// TIA Portal V18 export
FUNCTION_BLOCK "Stacklight"   // FB20, LAD
TITLE = Description:
{ S7_Optimized_Access := 'TRUE' }
VERSION : 0.1
// The stacklight is showing the status of the machine and checking different conditions:
// - errors from the drives (PLC)
// - communication (NOAH)
// - errors from the fluid supply (NOAH)
// - doors (PLC)
// 
// RED - default color, error or PLC is turning on
// ORANGE - door open or in maintenance mode
// GREEN - machine connected and working fine
// 
// RED-GREEN blinking - machine ready to connect
// 
// Date:
// stored: AutoNumber true, IsIECCheckEnabled false, IsRetainMemResEnabled false, MemoryReserve 100, SetENOAutomatically false, UDAEnableTagReadback false
   VAR_INPUT
      Emergency : Bool;
      Mode : Int;
      RedIn : Bool;
      YellowIn : Bool;
      GreenIn : Bool;
      ReadyDevices : Bool;
      DoorOpen : Bool;
      Xvelocity : DInt;
      Yvelocity : DInt;
      MachineReadyPLC : Bool;
      MachineReadyNOAH : Bool;
      MachinePrintingPLC : Bool;
      MachinePrintingNOAH : Bool;
      MachineErrorPLC : Bool;
      MachineErrorNOAH : Bool;
      LED01 : Bool;
      LED02 : Bool;
      Maintenance : Int;
   END_VAR
   VAR_OUTPUT
      Status : Int;
      OutputColor : Int;
      StacklightCTRL01 : Bool;
      StacklightCTRL02 : Bool;
   END_VAR
   VAR_IN_OUT
      MachineConnectedNOAH : Bool;
   END_VAR
   VAR
      TriggerVelocityForMoving : DInt := 5;
      GreenInternal : Bool;
      YellowInternal : Bool;
      RedInternal : Bool;
      ColorInternal : Int;   // 0 = Red; 1 = Orange; 2 = Green;
      MachineMovingInternal : Bool;
      MachineConnectedPLC : Bool;
      MachineConnectedInternal : Bool;
   END_VAR
   VAR CONSTANT
      MachineConnectedWaitTime : Time := T#3s;
      MachineConnectedResetTime : Time := T#200ms;
   END_VAR
BEGIN

REGION Network 1: Machine Moving Status Read
   // Checking if the machine is moving.
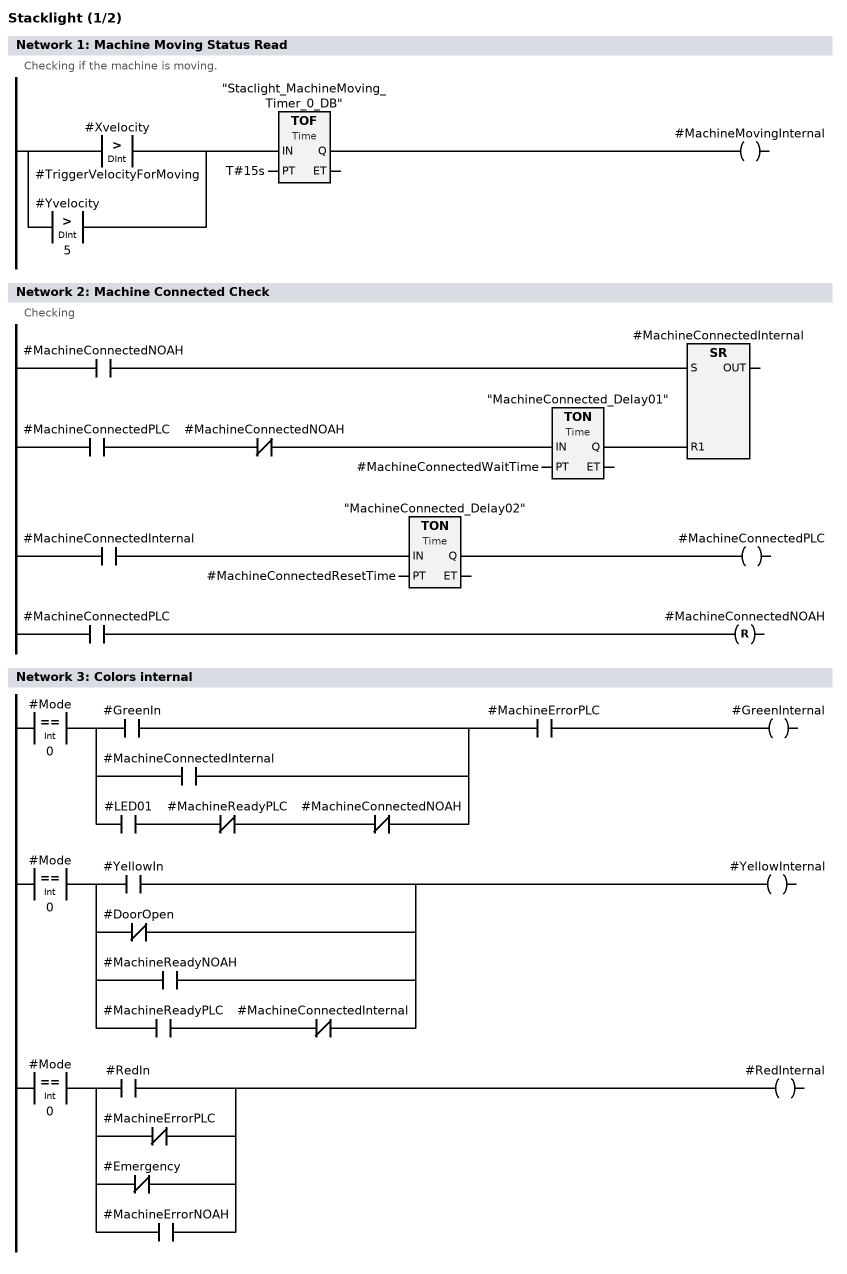
   RUNG wire#powerrail
      { S7_Templates := "SrcType := DInt" } GT_Contact(in1 := #Xvelocity, in2 := #TriggerVelocityForMoving)
      wire#w1
      { S7_Templates := "time_type := Time" } "Staclight_MachineMoving_Timer_0_DB".TOF(pt := T#15s, et =>)
      Coil( #MachineMovingInternal )
   END_RUNG
   RUNG wire#powerrail
      { S7_Templates := "SrcType := DInt" } GT_Contact(in1 := #Yvelocity, in2 := 5)
   END_RUNG wire#w1
   // the same network as SCL:
   "Staclight_MachineMoving_Timer_0_DB".TOF(IN := (#Xvelocity > #TriggerVelocityForMoving) OR (#Yvelocity > 5),
                           PT := T#15s);
   #MachineMovingInternal := "Staclight_MachineMoving_Timer_0_DB".Q;
END_REGION

REGION Network 2: Machine Connected Check
   // Checking
   RUNG wire#powerrail
      Contact( #MachineConnectedNOAH )
      S_SR(operand := #MachineConnectedInternal, r1 := wire#w1)
   END_RUNG
   RUNG wire#powerrail
      Contact( #MachineConnectedPLC )
      I_Contact( #MachineConnectedNOAH )
      { S7_Templates := "time_type := Time" } "MachineConnected_Delay01".TON(pt := #MachineConnectedWaitTime, et =>)
   END_RUNG wire#w1
   RUNG wire#powerrail
      Contact( #MachineConnectedInternal )
      { S7_Templates := "time_type := Time" } "MachineConnected_Delay02".TON(pt := #MachineConnectedResetTime, et =>)
      Coil( #MachineConnectedPLC )
   END_RUNG
   RUNG wire#powerrail
      Contact( #MachineConnectedPLC )
      R_Coil( #MachineConnectedNOAH )
   END_RUNG
   // the same network as SCL:
   "MachineConnected_Delay01".TON(IN := #MachineConnectedPLC AND NOT #MachineConnectedNOAH,
                           PT := #MachineConnectedWaitTime);
   IF #MachineConnectedNOAH THEN
       #MachineConnectedInternal := TRUE;   // SR flip-flop
   END_IF;
   IF "MachineConnected_Delay01".Q THEN #MachineConnectedInternal := FALSE; END_IF;
   "MachineConnected_Delay02".TON(IN := #MachineConnectedInternal, PT := #MachineConnectedResetTime);
   #MachineConnectedPLC := "MachineConnected_Delay02".Q;
   IF #MachineConnectedPLC THEN #MachineConnectedNOAH := FALSE; END_IF;
END_REGION

REGION Network 3: Colors internal
   RUNG wire#powerrail
      { S7_Templates := "SrcType := Int" } EQ_Contact(in1 := #Mode, in2 := 0)
      wire#w1
      Contact( #GreenIn )
      wire#w2
      Contact( #MachineErrorPLC )
      Coil( #GreenInternal )
   END_RUNG
   RUNG wire#w1
      Contact( #MachineConnectedInternal )
   END_RUNG wire#w2
   RUNG wire#w1
      Contact( #LED01 )
      I_Contact( #MachineReadyPLC )
      I_Contact( #MachineConnectedNOAH )
   END_RUNG wire#w2
   RUNG wire#powerrail
      { S7_Templates := "SrcType := Int" } EQ_Contact(in1 := #Mode, in2 := 0)
      wire#w3
      Contact( #YellowIn )
      wire#w4
      Coil( #YellowInternal )
   END_RUNG
   RUNG wire#w3
      I_Contact( #DoorOpen )
   END_RUNG wire#w4
   RUNG wire#w3
      Contact( #MachineReadyNOAH )
   END_RUNG wire#w4
   RUNG wire#w3
      Contact( #MachineReadyPLC )
      I_Contact( #MachineConnectedInternal )
   END_RUNG wire#w4
   RUNG wire#powerrail
      { S7_Templates := "SrcType := Int" } EQ_Contact(in1 := #Mode, in2 := 0)
      wire#w5
      Contact( #RedIn )
      wire#w6
      Coil( #RedInternal )
   END_RUNG
   RUNG wire#w5
      I_Contact( #MachineErrorPLC )
   END_RUNG wire#w6
   RUNG wire#w5
      I_Contact( #Emergency )
   END_RUNG wire#w6
   RUNG wire#w5
      Contact( #MachineErrorNOAH )
   END_RUNG wire#w6
   // the same network as SCL:
   #GreenInternal := (#Mode = 0) AND (#GreenIn OR #MachineConnectedInternal OR (#LED01 AND NOT #MachineReadyPLC AND NOT #MachineConnectedNOAH)) AND #MachineErrorPLC;
   #YellowInternal := (#Mode = 0) AND (#YellowIn OR NOT #DoorOpen OR #MachineReadyNOAH OR (#MachineReadyPLC AND NOT #MachineConnectedInternal));
   #RedInternal := (#Mode = 0) AND (#RedIn OR NOT #MachineErrorPLC OR NOT #Emergency OR #MachineErrorNOAH);
END_REGION

REGION Network 4: Status Move
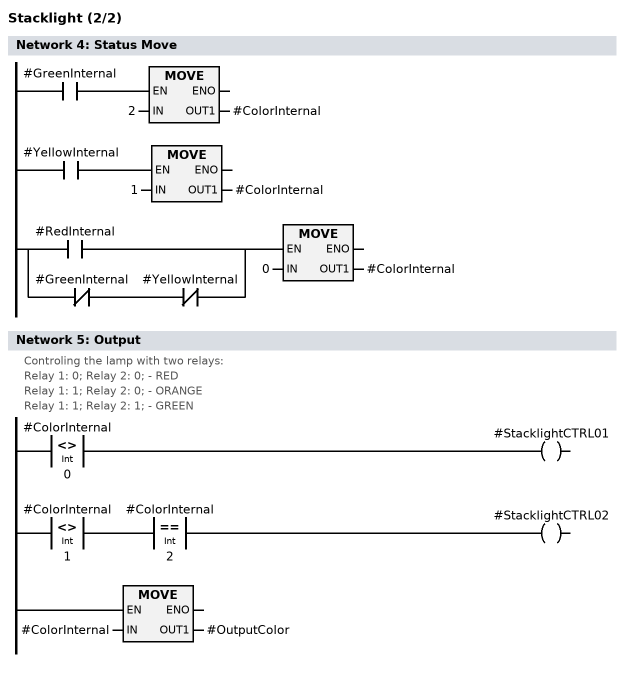
   RUNG wire#powerrail
      Contact( #GreenInternal )
      Move(in := 2, out1 => #ColorInternal)
   END_RUNG
   RUNG wire#powerrail
      Contact( #YellowInternal )
      Move(in := 1, out1 => #ColorInternal)
   END_RUNG
   RUNG wire#powerrail
      Contact( #RedInternal )
      wire#w1
      Move(in := 0, out1 => #ColorInternal)
   END_RUNG
   RUNG wire#powerrail
      I_Contact( #GreenInternal )
      I_Contact( #YellowInternal )
   END_RUNG wire#w1
   // the same network as SCL:
   IF #GreenInternal THEN #ColorInternal := 2; END_IF;
   IF #YellowInternal THEN #ColorInternal := 1; END_IF;
   IF #RedInternal OR (NOT #GreenInternal AND NOT #YellowInternal) THEN #ColorInternal := 0; END_IF;
END_REGION

REGION Network 5: Output
   // Controling the lamp with two relays:
   // Relay 1: 0; Relay 2: 0; - RED
   // Relay 1: 1; Relay 2: 0; - ORANGE
   // Relay 1: 1; Relay 2: 1; - GREEN
   RUNG wire#powerrail
      { S7_Templates := "SrcType := Int" } NE_Contact(in1 := #ColorInternal, in2 := 0)
      Coil( #StacklightCTRL01 )
   END_RUNG
   RUNG wire#powerrail
      { S7_Templates := "SrcType := Int" } NE_Contact(in1 := #ColorInternal, in2 := 1)
      { S7_Templates := "SrcType := Int" } EQ_Contact(in1 := #ColorInternal, in2 := 2)
      Coil( #StacklightCTRL02 )
   END_RUNG
   RUNG wire#powerrail
      Move(in := #ColorInternal, out1 => #OutputColor)
   END_RUNG
   // the same network as SCL:
   #StacklightCTRL01 := #ColorInternal <> 0;
   #StacklightCTRL02 := (#ColorInternal <> 1) AND (#ColorInternal = 2);
   #OutputColor := #ColorInternal;
END_REGION
END_FUNCTION_BLOCK
